LIN {X 0,Y 94.79,Z 775.203,A -85,B 0,C 180,E1 3730.047,E2 3730.047} C_VEL
LIN {X 0,Y 85.286,Z 779.428,A -85,B 0,C 180,E1 3718.728,E2 3718.728} C_VEL
LIN {X 0,Y 79.196,Z 781.917,A -85,B 0,C 180,E1 3705.374,E2 3705.374} C_VEL
LIN {X 0,Y 77.022,Z 782.778,A -85,B 0,C 180,E1 3690.744,E2 3690.744} C_VEL
LIN {X 0,Y 78.595,Z 782.144,A -85,B 0,C 180,E1 3676.763,E2 3676.763} C_VEL
LIN {X 0,Y 84.097,Z 779.929,A -85,B 0,C 180,E1 3663.142,E2 3663.142} C_VEL
LIN {X 0,Y 93.116,Z 776.003,A -85,B 0,C 180,E1 3651.481,E2 3651.481} C_VEL
LIN {X 0,Y 104.314,Z 770.552,A -85,B 0,C 180,E1 3642.436,E2 3642.436} C_VEL
LIN {X 0,Y 117.401,Z 763.276,A -85,B 0,C 180,E1 3635.158,E2 3635.158} C_VEL
LIN {X 0,Y 131.069,Z 754.49,A -85,B 0,C 180,E1 3629.586,E2 3629.586} C_VEL
LIN {X 0,Y 145.656,Z 743.569,A -85,B 0,C 180,E1 3625.03,E2 3625.03} C_VEL
LIN {X 0,Y 159.184,Z 731.747,A -85,B 0,C 180,E1 3621.631,E2 3621.631} C_VEL
LIN {X 0,Y 172.242,Z 718.44,A -85,B 0,C 180,E1 3618.884,E2 3618.884} C_VEL
LIN {X 0,Y 184.101,Z 704.311,A -85,B 0,C 180,E1 3616.73,E2 3616.73} C_VEL
LIN {X 0,Y 195.07,Z 688.928,A -85,B 0,C 180,E1 3614.95,E2 3614.95} C_VEL
LIN {X 0,Y 205.1,Z 672.108,A -85,B 0,C 180,E1 3613.461,E2 3613.461} C_VEL
LIN {X 0,Y 213.82,Z 654.238,A -85,B 0,C 180,E1 3612.234,E2 3612.234} C_VEL
LIN {X 0,Y 220.959,Z 635.839,A -85,B 0,C 180,E1 3611.251,E2 3611.251} C_VEL
LIN {X 0,Y 226.74,Z 615.995,A -85,B 0,C 180,E1 3610.436,E2 3610.436} C_VEL
LIN {X 0,Y 230.757,Z 595.786,A -85,B 0,C 180,E1 3609.81,E2 3609.81} C_VEL
LIN {X 0,Y 236.026,Z 551.57,A -85,B 0,C 180,E1 3608.94,E2 3608.94} C_VEL
LIN {X 0,Y 238.75,Z 528.075,A -85,B 0,C 180,E1 3608.563,E2 3608.563} C_VEL
LIN {X 0,Y 238.273,Z 526.572,A -85,B 0,C 180,E1 3606.506,E2 3606.506} C_VEL
LIN {X 0,Y 237.888,Z 526.562,A -85,B 0,C 180,E1 3602.168,E2 3602.168} C_VEL
LIN {X 0,Y 238.215,Z 528.774,A -85,B 0,C 180,E1 3598.918,E2 3598.918} C_VEL
LIN {X 0,Y 238.522,Z 530.833,A -85,B 0,C 180,E1 3597.356,E2 3597.356} C_VEL
LIN {X 0,Y 229.693,Z 603.415,A -85,B 0,C 180,E1 3596.168,E2 3596.168} C_VEL
LIN {X 0,Y 225.268,Z 624.242,A -85,B 0,C 180,E1 3595.75,E2 3595.75} C_VEL
LIN {X 0,Y 219.212,Z 644.095,A -85,B 0,C 180,E1 3595.261,E2 3595.261} C_VEL
LIN {X 0,Y 211.383,Z 663.553,A -85,B 0,C 180,E1 3594.655,E2 3594.655} C_VEL
LIN {X 0,Y 202.115,Z 681.945,A -85,B 0,C 180,E1 3593.885,E2 3593.885} C_VEL
LIN {X 0,Y 190.896,Z 700.299,A -85,B 0,C 180,E1 3592.779,E2 3592.779} C_VEL
LIN {X 0,Y 178.447,Z 717.368,A -85,B 0,C 180,E1 3591.299,E2 3591.299} C_VEL
LIN {X 0,Y 164.832,Z 733.27,A -85,B 0,C 180,E1 3589.311,E2 3589.311} C_VEL
LIN {X 0,Y 150.054,Z 748.089,A -85,B 0,C 180,E1 3586.61,E2 3586.61} C_VEL
LIN {X 0,Y 134.86,Z 761.302,A -85,B 0,C 180,E1 3583.016,E2 3583.016} C_VEL
LIN {X 0,Y 119.586,Z 772.97,A -85,B 0,C 180,E1 3578.131,E2 3578.131} C_VEL
LIN {X 0,Y 104.755,Z 783.066,A -85,B 0,C 180,E1 3571.412,E2 3571.412} C_VEL
LIN {X 0,Y 91.293,Z 791.543,A -85,B 0,C 180,E1 3562.049,E2 3562.049} C_VEL
LIN {X 0,Y 81.046,Z 798.03,A -85,B 0,C 180,E1 3549.904,E2 3549.904} C_VEL
LIN {X 0,Y 77.511,Z 800.568,A -85,B 0,C 180,E1 3542.778,E2 3542.778} C_VEL
LIN {X 0,Y 74.757,Z 801.989,A -85,B 0,C 180,E1 3537.407,E2 3537.407} C_VEL
LIN {X 0,Y 68.448,Z 803.712,A -85,B 0,C 180,E1 3525.965,E2 3525.965} C_VEL
LIN {X 0,Y 66.797,Z 804.343,A -85,B 0,C 180,E1 3518.037,E2 3518.037} C_VEL
LIN {X 0,Y 66.981,Z 804.481,A -85,B 0,C 180,E1 3515.654,E2 3515.654} C_VEL
LIN {X 0,Y 67.99,Z 804.819,A -85,B 0,C 180,E1 3509.63,E2 3509.63} C_VEL
LIN {X 0,Y 66.248,Z 803.424,A -85,B 0,C 180,E1 3494.237,E2 3494.237} C_VEL
LIN {X 0,Y 69.077,Z 800.295,A -85,B 0,C 180,E1 3477.619,E2 3477.619} C_VEL
LIN {X 0,Y 77.372,Z 795.212,A -85,B 0,C 180,E1 3462.559,E2 3462.559} C_VEL
LIN {X 0,Y 89.824,Z 788.216,A -85,B 0,C 180,E1 3451.009,E2 3451.009} C_VEL
LIN {X 0,Y 104.215,Z 779.674,A -85,B 0,C 180,E1 3442.924,E2 3442.924} C_VEL
LIN {X 0,Y 119.332,Z 769.699,A -85,B 0,C 180,E1 3437.223,E2 3437.223} C_VEL
LIN {X 0,Y 134.489,Z 758.36,A -85,B 0,C 180,E1 3433.12,E2 3433.12} C_VEL
LIN {X 0,Y 149.29,Z 745.693,A -85,B 0,C 180,E1 3430.102,E2 3430.102} C_VEL
LIN {X 0,Y 163.502,Z 731.675,A -85,B 0,C 180,E1 3427.843,E2 3427.843} C_VEL
LIN {X 0,Y 176.979,Z 716.205,A -85,B 0,C 180,E1 3426.12,E2 3426.12} C_VEL
LIN {X 0,Y 189.635,Z 699.109,A -85,B 0,C 180,E1 3424.808,E2 3424.808} C_VEL
LIN {X 0,Y 200.918,Z 680.865,A -85,B 0,C 180,E1 3423.846,E2 3423.846} C_VEL
LIN {X 0,Y 210.287,Z 662.45,A -85,B 0,C 180,E1 3423.175,E2 3423.175} C_VEL
LIN {X 0,Y 218.195,Z 642.954,A -85,B 0,C 180,E1 3422.643,E2 3422.643} C_VEL
LIN {X 0,Y 224.532,Z 622.209,A -85,B 0,C 180,E1 3422.192,E2 3422.192} C_VEL
LIN {X 0,Y 228.935,Z 601.111,A -85,B 0,C 180,E1 3421.809,E2 3421.809} C_VEL
LIN {X 0,Y 236.861,Z 536.432,A -85,B 0,C 180,E1 3420.801,E2 3420.801} C_VEL
LIN {X 0,Y 236.592,Z 534.278,A -85,B 0,C 180,E1 3417.82,E2 3417.82} C_VEL
LIN {X 0,Y 236.945,Z 534.241,A -85,B 0,C 180,E1 3413.701,E2 3413.701} C_VEL
LIN {X 0,Y 237.048,Z 534.547,A -85,B 0,C 180,E1 3413.152,E2 3413.152} C_VEL
LIN {X 0,Y 230.307,Z 591.088,A -85,B 0,C 180,E1 3412.191,E2 3412.191} C_VEL
LIN {X 0,Y 226.826,Z 610.801,A -85,B 0,C 180,E1 3411.658,E2 3411.658} C_VEL
LIN {X 0,Y 221.942,Z 629.319,A -85,B 0,C 180,E1 3411.006,E2 3411.006} C_VEL
LIN {X 0,Y 215.515,Z 647.484,A -85,B 0,C 180,E1 3410.187,E2 3410.187} C_VEL
LIN {X 0,Y 207.188,Z 665.867,A -85,B 0,C 180,E1 3409.123,E2 3409.123} C_VEL
LIN {X 0,Y 197.405,Z 683.311,A -85,B 0,C 180,E1 3407.829,E2 3407.829} C_VEL
LIN {X 0,Y 186.314,Z 699.654,A -85,B 0,C 180,E1 3406.243,E2 3406.243} C_VEL
LIN {X 0,Y 173.527,Z 715.411,A -85,B 0,C 180,E1 3404.201,E2 3404.201} C_VEL
LIN {X 0,Y 160.047,Z 729.424,A -85,B 0,C 180,E1 3401.724,E2 3401.724} C_VEL
LIN {X 0,Y 145.999,Z 741.842,A -85,B 0,C 180,E1 3398.647,E2 3398.647} C_VEL
LIN {X 0,Y 131.542,Z 752.736,A -85,B 0,C 180,E1 3394.756,E2 3394.756} C_VEL
LIN {X 0,Y 116.962,Z 762.108,A -85,B 0,C 180,E1 3389.699,E2 3389.699} C_VEL
LIN {X 0,Y 102.702,Z 769.932,A -85,B 0,C 180,E1 3382.967,E2 3382.967} C_VEL
LIN {X 0,Y 89.463,Z 776.145,A -85,B 0,C 180,E1 3373.861,E2 3373.861} C_VEL
LIN {X 0,Y 78.868,Z 780.452,A -85,B 0,C 180,E1 3362.171,E2 3362.171} C_VEL
LIN {X 0,Y 71.832,Z 783.018,A -85,B 0,C 180,E1 3347.832,E2 3347.832} C_VEL
LIN {X 0,Y 69.156,Z 783.937,A -85,B 0,C 180,E1 3332.486,E2 3332.486} C_VEL
LIN {X 0,Y 70.527,Z 783.466,A -85,B 0,C 180,E1 3316.89,E2 3316.89} C_VEL
LIN {X 0,Y 76.303,Z 781.422,A -85,B 0,C 180,E1 3301.854,E2 3301.854} C_VEL
LIN {X 0,Y 85.91,Z 777.677,A -85,B 0,C 180,E1 3289.328,E2 3289.328} C_VEL
LIN {X 0,Y 98.445,Z 772.088,A -85,B 0,C 180,E1 3279.478,E2 3279.478} C_VEL
LIN {X 0,Y 112.253,Z 764.919,A -85,B 0,C 180,E1 3272.204,E2 3272.204} C_VEL
LIN {X 0,Y 126.523,Z 756.253,A -85,B 0,C 180,E1 3266.752,E2 3266.752} C_VEL
LIN {X 0,Y 140.772,Z 746.14,A -85,B 0,C 180,E1 3262.584,E2 3262.584} C_VEL
LIN {X 0,Y 154.677,Z 734.619,A -85,B 0,C 180,E1 3259.311,E2 3259.311} C_VEL
LIN {X 0,Y 168.049,Z 721.668,A -85,B 0,C 180,E1 3256.687,E2 3256.687} C_VEL
LIN {X 0,Y 180.762,Z 707.191,A -85,B 0,C 180,E1 3254.543,E2 3254.543} C_VEL
LIN {X 0,Y 192.724,Z 690.993,A -85,B 0,C 180,E1 3252.756,E2 3252.756} C_VEL
LIN {X 0,Y 202.946,Z 674.402,A -85,B 0,C 180,E1 3251.366,E2 3251.366} C_VEL
LIN {X 0,Y 211.824,Z 656.824,A -85,B 0,C 180,E1 3250.219,E2 3250.219} C_VEL
LIN {X 0,Y 219.327,Z 638.171,A -85,B 0,C 180,E1 3249.269,E2 3249.269} C_VEL
LIN {X 0,Y 225.338,Z 618.422,A -85,B 0,C 180,E1 3248.491,E2 3248.491} C_VEL
LIN {X 0,Y 229.599,Z 598.14,A -85,B 0,C 180,E1 3247.882,E2 3247.882} C_VEL
LIN {X 0,Y 234.631,Z 557.443,A -85,B 0,C 180,E1 3247.085,E2 3247.085} C_VEL
LIN {X 0,Y 237.333,Z 534.597,A -85,B 0,C 180,E1 3246.714,E2 3246.714} C_VEL
LIN {X 0,Y 236.89,Z 534.461,A -85,B 0,C 180,E1 3242.42,E2 3242.42} C_VEL
LIN {X 0,Y 237.097,Z 536.385,A -85,B 0,C 180,E1 3239.517,E2 3239.517} C_VEL
LIN {X 0,Y 237.127,Z 536.857,A -85,B 0,C 180,E1 3239.187,E2 3239.187} C_VEL
LIN {X 0,Y 228.983,Z 602.568,A -85,B 0,C 180,E1 3238.174,E2 3238.174} C_VEL
LIN {X 0,Y 224.534,Z 623.283,A -85,B 0,C 180,E1 3237.795,E2 3237.795} C_VEL
LIN {X 0,Y 218.444,Z 643.068,A -85,B 0,C 180,E1 3237.363,E2 3237.363} C_VEL
LIN {X 0,Y 210.782,Z 661.997,A -85,B 0,C 180,E1 3236.851,E2 3236.851} C_VEL
LIN {X 0,Y 200.92,Z 681.371,A -85,B 0,C 180,E1 3236.147,E2 3236.147} C_VEL
LIN {X 0,Y 189.637,Z 699.509,A -85,B 0,C 180,E1 3235.184,E2 3235.184} C_VEL
LIN {X 0,Y 176.981,Z 716.533,A -85,B 0,C 180,E1 3233.873,E2 3233.873} C_VEL
LIN {X 0,Y 163.027,Z 732.455,A -85,B 0,C 180,E1 3232.081,E2 3232.081} C_VEL
LIN {X 0,Y 148.356,Z 746.799,A -85,B 0,C 180,E1 3229.72,E2 3229.72} C_VEL
LIN {X 0,Y 132.674,Z 760.024,A -85,B 0,C 180,E1 3226.444,E2 3226.444} C_VEL
LIN {X 0,Y 116.739,Z 771.695,A -85,B 0,C 180,E1 3221.93,E2 3221.93} C_VEL
LIN {X 0,Y 101.029,Z 781.796,A -85,B 0,C 180,E1 3215.571,E2 3215.571} C_VEL
LIN {X 0,Y 86.409,Z 790.275,A -85,B 0,C 180,E1 3206.419,E2 3206.419} C_VEL
LIN {X 0,Y 74.612,Z 796.891,A -85,B 0,C 180,E1 3193.646,E2 3193.646} C_VEL
LIN {X 0,Y 67.665,Z 801.488,A -85,B 0,C 180,E1 3177.556,E2 3177.556} C_VEL
LIN {X 0,Y 66.421,Z 804.095,A -85,B 0,C 180,E1 3160.407,E2 3160.407} C_VEL
LIN {X 0,Y 66.981,Z 804.481,A -85,B 0,C 180,E1 3155.654,E2 3155.654} C_VEL
LIN {X 0,Y 66.693,Z 804.571,A -85,B 0,C 180,E1 3152.598,E2 3152.598} C_VEL
LIN {X 0,Y 64.66,Z 804.284,A -85,B 0,C 180,E1 3148.461,E2 3148.461} C_VEL
LIN {X 0,Y 58.75,Z 802.884,A -85,B 0,C 180,E1 3138.157,E2 3138.157} C_VEL
LIN {X 0,Y 58.309,Z 802.507,A -85,B 0,C 180,E1 3135.107,E2 3135.107} C_VEL
LIN {X 0,Y 61.542,Z 799.446,A -85,B 0,C 180,E1 3115.346,E2 3115.346} C_VEL
LIN {X 0,Y 70.802,Z 794.549,A -85,B 0,C 180,E1 3099.042,E2 3099.042} C_VEL
LIN {X 0,Y 83.558,Z 788.148,A -85,B 0,C 180,E1 3087.692,E2 3087.692} C_VEL
LIN {X 0,Y 99.129,Z 779.667,A -85,B 0,C 180,E1 3079.441,E2 3079.441} C_VEL
LIN {X 0,Y 115.328,Z 769.658,A -85,B 0,C 180,E1 3073.838,E2 3073.838} C_VEL
LIN {X 0,Y 130.975,Z 758.559,A -85,B 0,C 180,E1 3070.019,E2 3070.019} C_VEL
LIN {X 0,Y 147.104,Z 745.276,A -85,B 0,C 180,E1 3067.101,E2 3067.101} C_VEL
LIN {X 0,Y 162.096,Z 730.871,A -85,B 0,C 180,E1 3065.026,E2 3065.026} C_VEL
LIN {X 0,Y 176.293,Z 714.854,A -85,B 0,C 180,E1 3063.469,E2 3063.469} C_VEL
LIN {X 0,Y 189.126,Z 697.707,A -85,B 0,C 180,E1 3062.343,E2 3062.343} C_VEL
LIN {X 0,Y 200.04,Z 680.284,A -85,B 0,C 180,E1 3061.56,E2 3061.56} C_VEL
LIN {X 0,Y 209.496,Z 661.945,A -85,B 0,C 180,E1 3060.993,E2 3060.993} C_VEL
LIN {X 0,Y 217.523,Z 642.437,A -85,B 0,C 180,E1 3060.537,E2 3060.537} C_VEL
LIN {X 0,Y 223.931,Z 621.816,A -85,B 0,C 180,E1 3060.145,E2 3060.145} C_VEL
LIN {X 0,Y 228.431,Z 600.738,A -85,B 0,C 180,E1 3059.801,E2 3059.801} C_VEL
LIN {X 0,Y 235.632,Z 543.029,A -85,B 0,C 180,E1 3058.966,E2 3058.966} C_VEL
LIN {X 0,Y 235.593,Z 542.128,A -85,B 0,C 180,E1 3057.324,E2 3057.324} C_VEL
LIN {X 0,Y 235.733,Z 542.122,A -85,B 0,C 180,E1 3054.985,E2 3054.985} C_VEL
LIN {X 0,Y 229.443,Z 593.572,A -85,B 0,C 180,E1 3054.131,E2 3054.131} C_VEL
LIN {X 0,Y 225.559,Z 614.046,A -85,B 0,C 180,E1 3053.593,E2 3053.593} C_VEL
LIN {X 0,Y 220.134,Z 633.241,A -85,B 0,C 180,E1 3052.937,E2 3052.937} C_VEL
LIN {X 0,Y 212.981,Z 652.126,A -85,B 0,C 180,E1 3052.109,E2 3052.109} C_VEL
LIN {X 0,Y 204.421,Z 669.941,A -85,B 0,C 180,E1 3051.112,E2 3051.112} C_VEL
LIN {X 0,Y 194.523,Z 686.751,A -85,B 0,C 180,E1 3049.916,E2 3049.916} C_VEL
LIN {X 0,Y 183.19,Z 702.748,A -85,B 0,C 180,E1 3048.433,E2 3048.433} C_VEL
LIN {X 0,Y 170.616,Z 717.665,A -85,B 0,C 180,E1 3046.601,E2 3046.601} C_VEL
LIN {X 0,Y 157.746,Z 730.671,A -85,B 0,C 180,E1 3044.453,E2 3044.453} C_VEL
LIN {X 0,Y 143.306,Z 743.076,A -85,B 0,C 180,E1 3041.596,E2 3041.596} C_VEL
LIN {X 0,Y 128.363,Z 753.961,A -85,B 0,C 180,E1 3037.957,E2 3037.957} C_VEL
LIN {X 0,Y 113.169,Z 763.326,A -85,B 0,C 180,E1 3033.166,E2 3033.166} C_VEL
LIN {X 0,Y 97.751,Z 771.333,A -85,B 0,C 180,E1 3026.471,E2 3026.471} C_VEL
LIN {X 0,Y 83.271,Z 777.616,A -85,B 0,C 180,E1 3017.09,E2 3017.09} C_VEL
LIN {X 0,Y 71.46,Z 781.937,A -85,B 0,C 180,E1 3004.355,E2 3004.355} C_VEL
LIN {X 0,Y 63.8,Z 784.403,A -85,B 0,C 180,E1 2988.266,E2 2988.266} C_VEL
LIN {X 0,Y 61.2,Z 785.2,A -85,B 0,C 180,E1 2970,E2 2970} C_VEL
LIN {X 0,Y 63.781,Z 784.429,A -85,B 0,C 180,E1 2951.729,E2 2951.729} C_VEL
LIN {X 0,Y 71.262,Z 782.046,A -85,B 0,C 180,E1 2935.861,E2 2935.861} C_VEL
LIN {X 0,Y 82.576,Z 777.942,A -85,B 0,C 180,E1 2923.408,E2 2923.408} C_VEL
LIN {X 0,Y 95.818,Z 772.302,A -85,B 0,C 180,E1 2914.479,E2 2914.479} C_VEL
LIN {X 0,Y 109.848,Z 765.261,A -85,B 0,C 180,E1 2908.007,E2 2908.007} C_VEL
LIN {X 0,Y 124.866,Z 756.375,A -85,B 0,C 180,E1 2902.952,E2 2902.952} C_VEL
LIN {X 0,Y 139.694,Z 746.022,A -85,B 0,C 180,E1 2899.133,E2 2899.133} C_VEL
LIN {X 0,Y 154.055,Z 734.233,A -85,B 0,C 180,E1 2896.152,E2 2896.152} C_VEL
LIN {X 0,Y 167.795,Z 720.972,A -85,B 0,C 180,E1 2893.77,E2 2893.77} C_VEL
LIN {X 0,Y 180.342,Z 706.72,A -85,B 0,C 180,E1 2891.895,E2 2891.895} C_VEL
LIN {X 0,Y 191.484,Z 691.818,A -85,B 0,C 180,E1 2890.405,E2 2890.405} C_VEL
LIN {X 0,Y 201.999,Z 674.988,A -85,B 0,C 180,E1 2889.114,E2 2889.114} C_VEL
LIN {X 0,Y 211.047,Z 657.306,A -85,B 0,C 180,E1 2888.057,E2 2888.057} C_VEL
LIN {X 0,Y 218.915,Z 637.859,A -85,B 0,C 180,E1 2887.149,E2 2887.149} C_VEL
LIN {X 0,Y 224.94,Z 617.986,A -85,B 0,C 180,E1 2886.432,E2 2886.432} C_VEL
LIN {X 0,Y 229.184,Z 597.547,A -85,B 0,C 180,E1 2885.866,E2 2885.866} C_VEL
LIN {X 0,Y 234.66,Z 553.561,A -85,B 0,C 180,E1 2885.077,E2 2885.077} C_VEL
LIN {X 0,Y 236.022,Z 542.248,A -85,B 0,C 180,E1 2884.901,E2 2884.901} C_VEL
LIN {X 0,Y 235.911,Z 542.576,A -85,B 0,C 180,E1 2881.944,E2 2881.944} C_VEL
LIN {X 0,Y 235.906,Z 543.467,A -85,B 0,C 180,E1 2881.03,E2 2881.03} C_VEL
LIN {X 0,Y 228.524,Z 601.888,A -85,B 0,C 180,E1 2880.186,E2 2880.186} C_VEL
LIN {X 0,Y 224.052,Z 622.45,A -85,B 0,C 180,E1 2879.848,E2 2879.848} C_VEL
LIN {X 0,Y 217.921,Z 642.174,A -85,B 0,C 180,E1 2879.475,E2 2879.475} C_VEL
LIN {X 0,Y 209.994,Z 661.529,A -85,B 0,C 180,E1 2879.027,E2 2879.027} C_VEL
LIN {X 0,Y 200.538,Z 679.92,A -85,B 0,C 180,E1 2878.464,E2 2878.464} C_VEL
LIN {X 0,Y 189.127,Z 698.131,A -85,B 0,C 180,E1 2877.649,E2 2877.649} C_VEL
LIN {X 0,Y 176.294,Z 715.199,A -85,B 0,C 180,E1 2876.523,E2 2876.523} C_VEL
LIN {X 0,Y 162.585,Z 730.642,A -85,B 0,C 180,E1 2875.025,E2 2875.025} C_VEL
LIN {X 0,Y 147.106,Z 745.507,A -85,B 0,C 180,E1 2872.891,E2 2872.891} C_VEL
LIN {X 0,Y 130.978,Z 758.744,A -85,B 0,C 180,E1 2869.975,E2 2869.975} C_VEL
LIN {X 0,Y 114.43,Z 770.421,A -85,B 0,C 180,E1 2865.897,E2 2865.897} C_VEL
LIN {X 0,Y 97.874,Z 780.525,A -85,B 0,C 180,E1 2860.022,E2 2860.022} C_VEL
LIN {X 0,Y 82.085,Z 789.006,A -85,B 0,C 180,E1 2851.282,E2 2851.282} C_VEL
LIN {X 0,Y 69.092,Z 795.5,A -85,B 0,C 180,E1 2838.806,E2 2838.806} C_VEL
LIN {X 0,Y 60.631,Z 800.105,A -85,B 0,C 180,E1 2821.849,E2 2821.849} C_VEL
LIN {X 0,Y 58.387,Z 802.851,A -85,B 0,C 180,E1 2801.858,E2 2801.858} C_VEL
LIN {X 0,Y 59.99,Z 803.61,A -85,B 0,C 180,E1 2789.92,E2 2789.92} C_VEL
LIN {X 0,Y 58.309,Z 802.507,A -85,B 0,C 180,E1 2775.107,E2 2775.107} C_VEL
LIN {X 0,Y 57.755,Z 801.514,A -85,B 0,C 180,E1 2767.524,E2 2767.524} C_VEL
LIN {X 0,Y 57.592,Z 797.296,A -85,B 0,C 180,E1 2746.102,E2 2746.102} C_VEL
LIN {X 0,Y 59.976,Z 795.854,A -85,B 0,C 180,E1 2740.775,E2 2740.775} C_VEL
LIN {X 0,Y 72.988,Z 790.122,A -85,B 0,C 180,E1 2727.075,E2 2727.075} C_VEL
LIN {X 0,Y 88.363,Z 782.767,A -85,B 0,C 180,E1 2718.11,E2 2718.11} C_VEL
LIN {X 0,Y 104.879,Z 773.742,A -85,B 0,C 180,E1 2712.106,E2 2712.106} C_VEL
LIN {X 0,Y 121.175,Z 763.407,A -85,B 0,C 180,E1 2708.053,E2 2708.053} C_VEL
LIN {X 0,Y 137.53,Z 751.311,A -85,B 0,C 180,E1 2705.139,E2 2705.139} C_VEL
LIN {X 0,Y 153.668,Z 737.323,A -85,B 0,C 180,E1 2702.983,E2 2702.983} C_VEL
LIN {X 0,Y 168.442,Z 722.251,A -85,B 0,C 180,E1 2701.454,E2 2701.454} C_VEL
LIN {X 0,Y 181.972,Z 705.964,A -85,B 0,C 180,E1 2700.349,E2 2700.349} C_VEL
LIN {X 0,Y 193.973,Z 688.764,A -85,B 0,C 180,E1 2699.563,E2 2699.563} C_VEL
LIN {X 0,Y 204.496,Z 670.555,A -85,B 0,C 180,E1 2699.006,E2 2699.006} C_VEL
LIN {X 0,Y 213.528,Z 651.227,A -85,B 0,C 180,E1 2698.59,E2 2698.59} C_VEL
LIN {X 0,Y 220.816,Z 631.121,A -85,B 0,C 180,E1 2698.242,E2 2698.242} C_VEL
LIN {X 0,Y 226.297,Z 610.268,A -85,B 0,C 180,E1 2697.927,E2 2697.927} C_VEL
LIN {X 0,Y 229.862,Z 588.948,A -85,B 0,C 180,E1 2697.629,E2 2697.629} C_VEL
LIN {X 0,Y 234.62,Z 550.029,A -85,B 0,C 180,E1 2697.068,E2 2697.068} C_VEL
LIN {X 0,Y 234.603,Z 550.172,A -85,B 0,C 180,E1 2696.831,E2 2696.831} C_VEL
LIN {X 0,Y 228.774,Z 596.534,A -85,B 0,C 180,E1 2696.072,E2 2696.072} C_VEL
LIN {X 0,Y 224.789,Z 616.292,A -85,B 0,C 180,E1 2695.574,E2 2695.574} C_VEL
LIN {X 0,Y 219.306,Z 634.998,A -85,B 0,C 180,E1 2694.974,E2 2694.974} C_VEL
LIN {X 0,Y 212.044,Z 653.683,A -85,B 0,C 180,E1 2694.214,E2 2694.214} C_VEL
LIN {X 0,Y 202.871,Z 672.256,A -85,B 0,C 180,E1 2693.253,E2 2693.253} C_VEL
LIN {X 0,Y 192.291,Z 689.613,A -85,B 0,C 180,E1 2692.104,E2 2692.104} C_VEL
LIN {X 0,Y 180.343,Z 705.825,A -85,B 0,C 180,E1 2690.695,E2 2690.695} C_VEL
LIN {X 0,Y 167.071,Z 720.899,A -85,B 0,C 180,E1 2688.948,E2 2688.948} C_VEL
LIN {X 0,Y 152.678,Z 734.658,A -85,B 0,C 180,E1 2686.749,E2 2686.749} C_VEL
LIN {X 0,Y 137.345,Z 747.003,A -85,B 0,C 180,E1 2683.929,E2 2683.929} C_VEL
LIN {X 0,Y 121.154,Z 757.938,A -85,B 0,C 180,E1 2680.185,E2 2680.185} C_VEL
LIN {X 0,Y 105.121,Z 766.97,A -85,B 0,C 180,E1 2675.258,E2 2675.258} C_VEL
LIN {X 0,Y 89.249,Z 774.383,A -85,B 0,C 180,E1 2668.365,E2 2668.365} C_VEL
LIN {X 0,Y 74.638,Z 780.002,A -85,B 0,C 180,E1 2658.604,E2 2658.604} C_VEL
LIN {X 0,Y 62.804,Z 783.772,A -85,B 0,C 180,E1 2644.968,E2 2644.968} C_VEL
LIN {X 0,Y 55.242,Z 785.846,A -85,B 0,C 180,E1 2626.833,E2 2626.833} C_VEL
LIN {X 0,Y 53.351,Z 786.348,A -85,B 0,C 180,E1 2606.777,E2 2606.777} C_VEL
LIN {X 0,Y 56.942,Z 785.467,A -85,B 0,C 180,E1 2587.276,E2 2587.276} C_VEL
LIN {X 0,Y 65.952,Z 782.941,A -85,B 0,C 180,E1 2570.453,E2 2570.453} C_VEL
LIN {X 0,Y 78.749,Z 778.667,A -85,B 0,C 180,E1 2558.078,E2 2558.078} C_VEL
LIN {X 0,Y 93.957,Z 772.498,A -85,B 0,C 180,E1 2549.24,E2 2549.24} C_VEL
LIN {X 0,Y 109.988,Z 764.604,A -85,B 0,C 180,E1 2543.011,E2 2543.011} C_VEL
LIN {X 0,Y 126.173,Z 754.999,A -85,B 0,C 180,E1 2538.481,E2 2538.481} C_VEL
LIN {X 0,Y 141.882,Z 743.858,A -85,B 0,C 180,E1 2535.11,E2 2535.11} C_VEL
LIN {X 0,Y 156.749,Z 731.349,A -85,B 0,C 180,E1 2532.526,E2 2532.526} C_VEL
LIN {X 0,Y 171.051,Z 717.058,A -85,B 0,C 180,E1 2530.441,E2 2530.441} C_VEL
LIN {X 0,Y 184.125,Z 701.487,A -85,B 0,C 180,E1 2528.778,E2 2528.778} C_VEL
LIN {X 0,Y 195.624,Z 685.09,A -85,B 0,C 180,E1 2527.464,E2 2527.464} C_VEL
LIN {X 0,Y 205.693,Z 667.69,A -85,B 0,C 180,E1 2526.389,E2 2526.389} C_VEL
LIN {X 0,Y 214.444,Z 648.925,A -85,B 0,C 180,E1 2525.481,E2 2525.481} C_VEL
LIN {X 0,Y 221.561,Z 629.164,A -85,B 0,C 180,E1 2524.733,E2 2524.733} C_VEL
LIN {X 0,Y 226.833,Z 608.925,A -85,B 0,C 180,E1 2524.135,E2 2524.135} C_VEL
LIN {X 0,Y 230.244,Z 588.417,A -85,B 0,C 180,E1 2523.668,E2 2523.668} C_VEL
LIN {X 0,Y 234.909,Z 550.241,A -85,B 0,C 180,E1 2523.05,E2 2523.05} C_VEL
LIN {X 0,Y 234.874,Z 550.537,A -85,B 0,C 180,E1 2522.885,E2 2522.885} C_VEL
LIN {X 0,Y 228.383,Z 601.024,A -85,B 0,C 180,E1 2522.206,E2 2522.206} C_VEL
LIN {X 0,Y 223.867,Z 621.585,A -85,B 0,C 180,E1 2521.909,E2 2521.909} C_VEL
LIN {X 0,Y 217.741,Z 641.16,A -85,B 0,C 180,E1 2521.596,E2 2521.596} C_VEL
LIN {X 0,Y 210.013,Z 659.968,A -85,B 0,C 180,E1 2521.24,E2 2521.24} C_VEL
LIN {X 0,Y 200.347,Z 678.704,A -85,B 0,C 180,E1 2520.778,E2 2520.778} C_VEL
LIN {X 0,Y 188.968,Z 696.743,A -85,B 0,C 180,E1 2520.12,E2 2520.12} C_VEL
LIN {X 0,Y 175.988,Z 713.859,A -85,B 0,C 180,E1 2519.186,E2 2519.186} C_VEL
LIN {X 0,Y 161.571,Z 729.855,A -85,B 0,C 180,E1 2517.873,E2 2517.873} C_VEL
LIN {X 0,Y 146.112,Z 744.389,A -85,B 0,C 180,E1 2516.077,E2 2516.077} C_VEL
LIN {X 0,Y 129.791,Z 757.463,A -85,B 0,C 180,E1 2513.583,E2 2513.583} C_VEL
LIN {X 0,Y 112.691,Z 769.146,A -85,B 0,C 180,E1 2510.004,E2 2510.004} C_VEL
LIN {X 0,Y 95.347,Z 779.255,A -85,B 0,C 180,E1 2504.738,E2 2504.738} C_VEL
LIN {X 0,Y 78.415,Z 787.738,A -85,B 0,C 180,E1 2496.64,E2 2496.64} C_VEL
LIN {X 0,Y 63.911,Z 794.235,A -85,B 0,C 180,E1 2484.438,E2 2484.438} C_VEL
LIN {X 0,Y 53.764,Z 798.845,A -85,B 0,C 180,E1 2466.519,E2 2466.519} C_VEL
LIN {X 0,Y 50.391,Z 801.627,A -85,B 0,C 180,E1 2443.538,E2 2443.538} C_VEL
LIN {X 0,Y 51.916,Z 802.384,A -85,B 0,C 180,E1 2430,E2 2430} C_VEL
LIN {X 0,Y 50.587,Z 800.922,A -85,B 0,C 180,E1 2409.16,E2 2409.16} C_VEL
LIN {X 0,Y 56.209,Z 797.564,A -85,B 0,C 180,E1 2387.473,E2 2387.473} C_VEL
LIN {X 0,Y 59.976,Z 795.854,A -85,B 0,C 180,E1 2380.775,E2 2380.775} C_VEL
LIN {X 0,Y 63.488,Z 793.944,A -85,B 0,C 180,E1 2374.597,E2 2374.597} C_VEL
LIN {X 0,Y 73.141,Z 787.653,A -85,B 0,C 180,E1 2359.522,E2 2359.522} C_VEL
LIN {X 0,Y 77.807,Z 785.332,A -85,B 0,C 180,E1 2356.368,E2 2356.368} C_VEL
LIN {X 0,Y 94.429,Z 777.363,A -85,B 0,C 180,E1 2350.037,E2 2350.037} C_VEL
LIN {X 0,Y 111.547,Z 767.711,A -85,B 0,C 180,E1 2345.775,E2 2345.775} C_VEL
LIN {X 0,Y 129.127,Z 755.981,A -85,B 0,C 180,E1 2342.751,E2 2342.751} C_VEL
LIN {X 0,Y 145.985,Z 742.671,A -85,B 0,C 180,E1 2340.653,E2 2340.653} C_VEL
LIN {X 0,Y 161.488,Z 728.226,A -85,B 0,C 180,E1 2339.199,E2 2339.199} C_VEL
LIN {X 0,Y 175.559,Z 712.766,A -85,B 0,C 180,E1 2338.173,E2 2338.173} C_VEL
LIN {X 0,Y 188.154,Z 696.372,A -85,B 0,C 180,E1 2337.452,E2 2337.452} C_VEL
LIN {X 0,Y 199.249,Z 679.077,A -85,B 0,C 180,E1 2336.947,E2 2336.947} C_VEL
LIN {X 0,Y 208.833,Z 660.918,A -85,B 0,C 180,E1 2336.594,E2 2336.594} C_VEL
LIN {X 0,Y 212.676,Z 652.363,A -85,B 0,C 180,E1 2336.453,E2 2336.453} C_VEL
LIN {X 0,Y 204.053,Z 670.181,A -85,B 0,C 180,E1 2335.652,E2 2335.652} C_VEL
LIN {X 0,Y 193.664,Z 687.596,A -85,B 0,C 180,E1 2334.667,E2 2334.667} C_VEL
LIN {X 0,Y 182.141,Z 703.588,A -85,B 0,C 180,E1 2333.496,E2 2333.496} C_VEL
LIN {X 0,Y 169.105,Z 718.73,A -85,B 0,C 180,E1 2332.031,E2 2332.031} C_VEL
LIN {X 0,Y 155.214,Z 732.323,A -85,B 0,C 180,E1 2330.254,E2 2330.254} C_VEL
LIN {X 0,Y 140.061,Z 744.825,A -85,B 0,C 180,E1 2327.954,E2 2327.954} C_VEL
LIN {X 0,Y 124.215,Z 755.806,A -85,B 0,C 180,E1 2324.995,E2 2324.995} C_VEL
LIN {X 0,Y 107.843,Z 765.272,A -85,B 0,C 180,E1 2321.025,E2 2321.025} C_VEL
LIN {X 0,Y 91.236,Z 773.187,A -85,B 0,C 180,E1 2315.447,E2 2315.447} C_VEL
LIN {X 0,Y 75.702,Z 779.207,A -85,B 0,C 180,E1 2307.702,E2 2307.702} C_VEL
LIN {X 0,Y 61.349,Z 783.693,A -85,B 0,C 180,E1 2295.814,E2 2295.814} C_VEL
LIN {X 0,Y 50.55,Z 786.423,A -85,B 0,C 180,E1 2278.34,E2 2278.34} C_VEL
LIN {X 0,Y 45.608,Z 787.501,A -85,B 0,C 180,E1 2256.293,E2 2256.293} C_VEL
LIN {X 0,Y 47.165,Z 787.194,A -85,B 0,C 180,E1 2232.736,E2 2232.736} C_VEL
LIN {X 0,Y 55.349,Z 785.326,A -85,B 0,C 180,E1 2212.108,E2 2212.108} C_VEL
LIN {X 0,Y 67.439,Z 782.004,A -85,B 0,C 180,E1 2198.209,E2 2198.209} C_VEL
LIN {X 0,Y 82.847,Z 776.709,A -85,B 0,C 180,E1 2188.239,E2 2188.239} C_VEL
LIN {X 0,Y 98.957,Z 769.858,A -85,B 0,C 180,E1 2181.638,E2 2181.638} C_VEL
LIN {X 0,Y 115.928,Z 761.002,A -85,B 0,C 180,E1 2176.799,E2 2176.799} C_VEL
LIN {X 0,Y 132.531,Z 750.496,A -85,B 0,C 180,E1 2173.296,E2 2173.296} C_VEL
LIN {X 0,Y 147.58,Z 739.153,A -85,B 0,C 180,E1 2170.78,E2 2170.78} C_VEL
LIN {X 0,Y 162.832,Z 725.464,A -85,B 0,C 180,E1 2168.668,E2 2168.668} C_VEL
LIN {X 0,Y 176.794,Z 710.501,A -85,B 0,C 180,E1 2167.017,E2 2167.017} C_VEL
LIN {X 0,Y 189.401,Z 694.329,A -85,B 0,C 180,E1 2165.691,E2 2165.691} C_VEL
LIN {X 0,Y 200.614,Z 676.933,A -85,B 0,C 180,E1 2164.607,E2 2164.607} C_VEL
LIN {X 0,Y 209.954,Z 659.194,A -85,B 0,C 180,E1 2163.74,E2 2163.74} C_VEL
LIN {X 0,Y 212.304,Z 653.923,A -85,B 0,C 180,E1 2163.519,E2 2163.519} C_VEL
LIN {X 0,Y 203.282,Z 672.394,A -85,B 0,C 180,E1 2163.202,E2 2163.202} C_VEL
LIN {X 0,Y 192.691,Z 690.076,A -85,B 0,C 180,E1 2162.762,E2 2162.762} C_VEL
LIN {X 0,Y 180.67,Z 706.774,A -85,B 0,C 180,E1 2162.133,E2 2162.133} C_VEL
LIN {X 0,Y 167.642,Z 722.073,A -85,B 0,C 180,E1 2161.274,E2 2161.274} C_VEL
LIN {X 0,Y 152.974,Z 736.714,A -85,B 0,C 180,E1 2160.04,E2 2160.04} C_VEL
LIN {X 0,Y 137.036,Z 750.232,A -85,B 0,C 180,E1 2158.303,E2 2158.303} C_VEL
LIN {X 0,Y 120.293,Z 762.301,A -85,B 0,C 180,E1 2155.86,E2 2155.86} C_VEL
LIN {X 0,Y 102.399,Z 773.217,A -85,B 0,C 180,E1 2152.144,E2 2152.144} C_VEL
LIN {X 0,Y 84.326,Z 782.486,A -85,B 0,C 180,E1 2146.471,E2 2146.471} C_VEL
LIN {X 0,Y 67.139,Z 789.96,A -85,B 0,C 180,E1 2137.413,E2 2137.413} C_VEL
LIN {X 0,Y 52.493,Z 795.592,A -85,B 0,C 180,E1 2122.449,E2 2122.449} C_VEL
LIN {X 0,Y 43.546,Z 799.345,A -85,B 0,C 180,E1 2098.827,E2 2098.827} C_VEL
LIN {X 0,Y 43.371,Z 801.043,A -85,B 0,C 180,E1 2072.642,E2 2072.642} C_VEL
LIN {X 0,Y 43.798,Z 801.151,A -85,B 0,C 180,E1 2070,E2 2070} C_VEL
LIN {X 0,Y 42.989,Z 799.656,A -85,B 0,C 180,E1 2045.099,E2 2045.099} C_VEL
LIN {X 0,Y 50.39,Z 796.299,A -85,B 0,C 180,E1 2021.063,E2 2021.063} C_VEL
LIN {X 0,Y 63.995,Z 791.093,A -85,B 0,C 180,E1 2004.949,E2 2004.949} C_VEL
LIN {X 0,Y 77.807,Z 785.332,A -85,B 0,C 180,E1 1996.368,E2 1996.368} C_VEL
LIN {X 0,Y 83.405,Z 782.539,A -85,B 0,C 180,E1 1993.103,E2 1993.103} C_VEL
LIN {X 0,Y 96.694,Z 774.657,A -85,B 0,C 180,E1 1984.844,E2 1984.844} C_VEL
LIN {X 0,Y 102.777,Z 771.132,A -85,B 0,C 180,E1 1982.957,E2 1982.957} C_VEL
LIN {X 0,Y 119.98,Z 760.841,A -85,B 0,C 180,E1 1980.179,E2 1980.179} C_VEL
LIN {X 0,Y 137.042,Z 748.732,A -85,B 0,C 180,E1 1978.227,E2 1978.227} C_VEL
LIN {X 0,Y 153.203,Z 735.16,A -85,B 0,C 180,E1 1976.867,E2 1976.867} C_VEL
LIN {X 0,Y 168.403,Z 720.049,A -85,B 0,C 180,E1 1975.895,E2 1975.895} C_VEL
LIN {X 0,Y 176.106,Z 711.289,A -85,B 0,C 180,E1 1975.477,E2 1975.477} C_VEL
LIN {X 0,Y 161.85,Z 726.387,A -85,B 0,C 180,E1 1974.033,E2 1974.033} C_VEL
LIN {X 0,Y 146.33,Z 740.113,A -85,B 0,C 180,E1 1972.197,E2 1972.197} C_VEL
LIN {X 0,Y 130.009,Z 752.149,A -85,B 0,C 180,E1 1969.86,E2 1969.86} C_VEL
LIN {X 0,Y 112.984,Z 762.559,A -85,B 0,C 180,E1 1966.761,E2 1966.761} C_VEL
LIN {X 0,Y 95.439,Z 771.333,A -85,B 0,C 180,E1 1962.425,E2 1962.425} C_VEL
LIN {X 0,Y 77.711,Z 778.429,A -85,B 0,C 180,E1 1955.992,E2 1955.992} C_VEL
LIN {X 0,Y 61.329,Z 783.568,A -85,B 0,C 180,E1 1946.248,E2 1946.248} C_VEL
LIN {X 0,Y 47.545,Z 786.903,A -85,B 0,C 180,E1 1930.686,E2 1930.686} C_VEL
LIN {X 0,Y 38.855,Z 788.556,A -85,B 0,C 180,E1 1906.443,E2 1906.443} C_VEL
LIN {X 0,Y 38.196,Z 788.652,A -85,B 0,C 180,E1 1877.913,E2 1877.913} C_VEL
LIN {X 0,Y 45.257,Z 787.359,A -85,B 0,C 180,E1 1853.382,E2 1853.382} C_VEL
LIN {X 0,Y 58.267,Z 784.401,A -85,B 0,C 180,E1 1836.246,E2 1836.246} C_VEL
LIN {X 0,Y 74.593,Z 779.556,A -85,B 0,C 180,E1 1825.402,E2 1825.402} C_VEL
LIN {X 0,Y 91.785,Z 773.007,A -85,B 0,C 180,E1 1818.611,E2 1818.611} C_VEL
LIN {X 0,Y 109.214,Z 764.709,A -85,B 0,C 180,E1 1813.974,E2 1813.974} C_VEL
LIN {X 0,Y 126.169,Z 754.817,A -85,B 0,C 180,E1 1810.692,E2 1810.692} C_VEL
LIN {X 0,Y 142.446,Z 743.362,A -85,B 0,C 180,E1 1808.24,E2 1808.24} C_VEL
LIN {X 0,Y 157.935,Z 730.32,A -85,B 0,C 180,E1 1806.328,E2 1806.328} C_VEL
LIN {X 0,Y 172.574,Z 715.584,A -85,B 0,C 180,E1 1804.792,E2 1804.792} C_VEL
LIN {X 0,Y 175.867,Z 711.955,A -85,B 0,C 180,E1 1804.476,E2 1804.476} C_VEL
LIN {X 0,Y 161.304,Z 727.727,A -85,B 0,C 180,E1 1803.673,E2 1803.673} C_VEL
LIN {X 0,Y 145.112,Z 742.471,A -85,B 0,C 180,E1 1802.493,E2 1802.493} C_VEL
LIN {X 0,Y 127.991,Z 755.597,A -85,B 0,C 180,E1 1800.809,E2 1800.809} C_VEL
LIN {X 0,Y 110.028,Z 767.168,A -85,B 0,C 180,E1 1798.333,E2 1798.333} C_VEL
LIN {X 0,Y 91.401,Z 777.171,A -85,B 0,C 180,E1 1794.527,E2 1794.527} C_VEL
LIN {X 0,Y 73.412,Z 785.202,A -85,B 0,C 180,E1 1788.694,E2 1788.694} C_VEL
LIN {X 0,Y 55.883,Z 791.703,A -85,B 0,C 180,E1 1778.489,E2 1778.489} C_VEL
LIN {X 0,Y 41.04,Z 796.501,A -85,B 0,C 180,E1 1759.045,E2 1759.045} C_VEL
LIN {X 0,Y 34.523,Z 799.286,A -85,B 0,C 180,E1 1727.121,E2 1727.121} C_VEL
LIN {X 0,Y 35.661,Z 799.914,A -85,B 0,C 180,E1 1710,E2 1710} C_VEL
LIN {X 0,Y 35.902,Z 798.299,A -85,B 0,C 180,E1 1678.053,E2 1678.053} C_VEL
LIN {X 0,Y 46.034,Z 794.827,A -85,B 0,C 180,E1 1652.107,E2 1652.107} C_VEL
LIN {X 0,Y 61.78,Z 789.533,A -85,B 0,C 180,E1 1637.284,E2 1637.284} C_VEL
LIN {X 0,Y 78.994,Z 782.724,A -85,B 0,C 180,E1 1629.158,E2 1629.158} C_VEL
LIN {X 0,Y 97.233,Z 774.068,A -85,B 0,C 180,E1 1624.101,E2 1624.101} C_VEL
LIN {X 0,Y 102.777,Z 771.132,A -85,B 0,C 180,E1 1622.957,E2 1622.957} C_VEL
LIN {X 0,Y 108.91,Z 767.484,A -85,B 0,C 180,E1 1621.302,E2 1621.302} C_VEL
LIN {X 0,Y 123.429,Z 757.685,A -85,B 0,C 180,E1 1616.388,E2 1616.388} C_VEL
LIN {X 0,Y 129.469,Z 753.349,A -85,B 0,C 180,E1 1615.395,E2 1615.395} C_VEL
LIN {X 0,Y 139.565,Z 745.837,A -85,B 0,C 180,E1 1614.64,E2 1614.64} C_VEL
LIN {X 0,Y 122.874,Z 757.133,A -85,B 0,C 180,E1 1612.518,E2 1612.518} C_VEL
LIN {X 0,Y 105.684,Z 766.726,A -85,B 0,C 180,E1 1609.704,E2 1609.704} C_VEL
LIN {X 0,Y 88.66,Z 774.461,A -85,B 0,C 180,E1 1605.892,E2 1605.892} C_VEL
LIN {X 0,Y 70.329,Z 781.056,A -85,B 0,C 180,E1 1599.766,E2 1599.766} C_VEL
LIN {X 0,Y 53.172,Z 785.723,A -85,B 0,C 180,E1 1589.879,E2 1589.879} C_VEL
LIN {X 0,Y 38.581,Z 788.624,A -85,B 0,C 180,E1 1572.361,E2 1572.361} C_VEL
LIN {X 0,Y 30.097,Z 789.884,A -85,B 0,C 180,E1 1541.498,E2 1541.498} C_VEL
LIN {X 0,Y 32.014,Z 789.659,A -85,B 0,C 180,E1 1506.046,E2 1506.046} C_VEL
LIN {X 0,Y 43.22,Z 787.88,A -85,B 0,C 180,E1 1480.235,E2 1480.235} C_VEL
LIN {X 0,Y 58.957,Z 784.417,A -85,B 0,C 180,E1 1466,E2 1466} C_VEL
LIN {X 0,Y 76.625,Z 779.126,A -85,B 0,C 180,E1 1457.726,E2 1457.726} C_VEL
LIN {X 0,Y 94.268,Z 772.282,A -85,B 0,C 180,E1 1452.637,E2 1452.637} C_VEL
LIN {X 0,Y 112.376,Z 763.438,A -85,B 0,C 180,E1 1449.037,E2 1449.037} C_VEL
LIN {X 0,Y 129.806,Z 752.952,A -85,B 0,C 180,E1 1446.476,E2 1446.476} C_VEL
LIN {X 0,Y 139.027,Z 746.499,A -85,B 0,C 180,E1 1445.314,E2 1445.314} C_VEL
LIN {X 0,Y 122.272,Z 758.394,A -85,B 0,C 180,E1 1443.965,E2 1443.965} C_VEL
LIN {X 0,Y 105.047,Z 768.698,A -85,B 0,C 180,E1 1442.011,E2 1442.011} C_VEL
LIN {X 0,Y 86.005,Z 778.161,A -85,B 0,C 180,E1 1438.764,E2 1438.764} C_VEL
LIN {X 0,Y 67.414,Z 785.69,A -85,B 0,C 180,E1 1433.559,E2 1433.559} C_VEL
LIN {X 0,Y 48.944,Z 791.712,A -85,B 0,C 180,E1 1423.763,E2 1423.763} C_VEL
LIN {X 0,Y 32.862,Z 796.042,A -85,B 0,C 180,E1 1402.282,E2 1402.282} C_VEL
LIN {X 0,Y 26.624,Z 798.324,A -85,B 0,C 180,E1 1362.486,E2 1362.486} C_VEL
LIN {X 0,Y 27.502,Z 798.675,A -85,B 0,C 180,E1 1350,E2 1350} C_VEL
LIN {X 0,Y 29.488,Z 796.969,A -85,B 0,C 180,E1 1308.236,E2 1308.236} C_VEL
LIN {X 0,Y 43.011,Z 793.354,A -85,B 0,C 180,E1 1281.589,E2 1281.589} C_VEL
LIN {X 0,Y 60.769,Z 787.961,A -85,B 0,C 180,E1 1269.182,E2 1269.182} C_VEL
LIN {X 0,Y 79.084,Z 781.053,A -85,B 0,C 180,E1 1262.849,E2 1262.849} C_VEL
LIN {X 0,Y 97.998,Z 772.289,A -85,B 0,C 180,E1 1259.022,E2 1259.022} C_VEL
LIN {X 0,Y 116.181,Z 762.063,A -85,B 0,C 180,E1 1256.634,E2 1256.634} C_VEL
LIN {X 0,Y 129.469,Z 753.349,A -85,B 0,C 180,E1 1255.395,E2 1255.395} C_VEL
LIN {X 0,Y 127.987,Z 754.261,A -85,B 0,C 180,E1 1254.947,E2 1254.947} C_VEL
LIN {X 0,Y 119.86,Z 759.395,A -85,B 0,C 180,E1 1254.356,E2 1254.356} C_VEL
LIN {X 0,Y 103.567,Z 768.51,A -85,B 0,C 180,E1 1254.171,E2 1254.171} C_VEL
LIN {X 0,Y 92.21,Z 774.105,A -85,B 0,C 180,E1 1254.891,E2 1254.891} C_VEL
LIN {X 0,Y 72.025,Z 782.574,A -85,B 0,C 180,E1 1258.157,E2 1258.157} C_VEL
LIN {X 0,Y 51.512,Z 789.275,A -85,B 0,C 180,E1 1264.451,E2 1264.451} C_VEL
LIN {X 0,Y 32.649,Z 793.94,A -85,B 0,C 180,E1 1278.318,E2 1278.318} C_VEL
LIN {X 0,Y 19.334,Z 796.785,A -85,B 0,C 180,E1 1318.859,E2 1318.859} C_VEL
LIN {X 0,Y 19.33,Z 797.434,A -85,B 0,C 180,E1 1349.999,E2 1349.999} C_VEL
LIN {X 0,Y 24.183,Z 795.689,A -85,B 0,C 180,E1 1405.779,E2 1405.779} C_VEL
LIN {X 0,Y 40.689,Z 792.136,A -85,B 0,C 180,E1 1429.387,E2 1429.387} C_VEL
LIN {X 0,Y 60.005,Z 786.763,A -85,B 0,C 180,E1 1438.711,E2 1438.711} C_VEL
LIN {X 0,Y 79.109,Z 779.885,A -85,B 0,C 180,E1 1443.191,E2 1443.191} C_VEL
LIN {X 0,Y 98.515,Z 771.143,A -85,B 0,C 180,E1 1445.826,E2 1445.826} C_VEL
LIN {X 0,Y 102.59,Z 769.098,A -85,B 0,C 180,E1 1446.241,E2 1446.241} C_VEL
LIN {X 0,Y 84.16,Z 776.957,A -85,B 0,C 180,E1 1449.583,E2 1449.583} C_VEL
LIN {X 0,Y 65.164,Z 783.216,A -85,B 0,C 180,E1 1454.846,E2 1454.846} C_VEL
LIN {X 0,Y 47.012,Z 787.573,A -85,B 0,C 180,E1 1463.865,E2 1463.865} C_VEL
LIN {X 0,Y 30.989,Z 790.177,A -85,B 0,C 180,E1 1482.092,E2 1482.092} C_VEL
LIN {X 0,Y 21.979,Z 791.134,A -85,B 0,C 180,E1 1519.516,E2 1519.516} C_VEL
LIN {X 0,Y 26.02,Z 790.716,A -85,B 0,C 180,E1 1565.197,E2 1565.197} C_VEL
LIN {X 0,Y 40.231,Z 788.736,A -85,B 0,C 180,E1 1590.438,E2 1590.438} C_VEL
LIN {X 0,Y 57.781,Z 785.064,A -85,B 0,C 180,E1 1602.122,E2 1602.122} C_VEL
LIN {X 0,Y 75.563,Z 779.885,A -85,B 0,C 180,E1 1608.28,E2 1608.28} C_VEL
LIN {X 0,Y 93.841,Z 772.906,A -85,B 0,C 180,E1 1612.253,E2 1612.253} C_VEL
LIN {X 0,Y 102.592,Z 768.942,A -85,B 0,C 180,E1 1613.754,E2 1613.754} C_VEL
LIN {X 0,Y 92.21,Z 774.105,A -85,B 0,C 180,E1 1614.891,E2 1614.891} C_VEL
LIN {X 0,Y 84.152,Z 777.602,A -85,B 0,C 180,E1 1615.308,E2 1615.308} C_VEL
LIN {X 0,Y 73.515,Z 781.417,A -85,B 0,C 180,E1 1614.359,E2 1614.359} C_VEL
LIN {X 0,Y 55.026,Z 786.476,A -85,B 0,C 180,E1 1609.629,E2 1609.629} C_VEL
LIN {X 0,Y 54.43,Z 786.622,A -85,B 0,C 180,E1 1609.434,E2 1609.434} C_VEL
LIN {X 0,Y 36.055,Z 790.087,A -85,B 0,C 180,E1 1600.537,E2 1600.537} C_VEL
LIN {X 0,Y 19.375,Z 791.979,A -85,B 0,C 180,E1 1576.259,E2 1576.259} C_VEL
LIN {X 0,Y 14.568,Z 792.315,A -85,B 0,C 180,E1 1509.932,E2 1509.932} C_VEL
LIN {X 0,Y 28.04,Z 791.175,A -85,B 0,C 180,E1 1466.946,E2 1466.946} C_VEL
LIN {X 0,Y 46.287,Z 788.398,A -85,B 0,C 180,E1 1453.582,E2 1453.582} C_VEL
LIN {X 0,Y 65.449,Z 783.885,A -85,B 0,C 180,E1 1447.462,E2 1447.462} C_VEL
LIN {X 0,Y 45.055,Z 789.688,A -85,B 0,C 180,E1 1443.031,E2 1443.031} C_VEL
LIN {X 0,Y 25.282,Z 793.681,A -85,B 0,C 180,E1 1431.374,E2 1431.374} C_VEL
LIN {X 0,Y 10.957,Z 795.875,A -85,B 0,C 180,E1 1377.146,E2 1377.146} C_VEL
LIN {X 0,Y 11.138,Z 796.189,A -85,B 0,C 180,E1 1349.999,E2 1349.999} C_VEL
LIN {X 0,Y 20.688,Z 794.409,A -85,B 0,C 180,E1 1274.854,E2 1274.854} C_VEL
LIN {X 0,Y 41.009,Z 790.615,A -85,B 0,C 180,E1 1258.387,E2 1258.387} C_VEL
LIN {X 0,Y 61.427,Z 785.12,A -85,B 0,C 180,E1 1253.161,E2 1253.161} C_VEL
LIN {X 0,Y 65.554,Z 783.757,A -85,B 0,C 180,E1 1252.476,E2 1252.476} C_VEL
LIN {X 0,Y 54.43,Z 786.622,A -85,B 0,C 180,E1 1249.434,E2 1249.434} C_VEL
LIN {X 0,Y 45.975,Z 788.577,A -85,B 0,C 180,E1 1247.472,E2 1247.472} C_VEL
LIN {X 0,Y 29.71,Z 791.568,A -85,B 0,C 180,E1 1246.261,E2 1246.261} C_VEL
LIN {X 0,Y 18.429,Z 792.943,A -85,B 0,C 180,E1 1242.637,E2 1242.637} C_VEL
LIN {X 0,Y 14.841,Z 793.195,A -85,B 0,C 180,E1 1238.285,E2 1238.285} C_VEL
LIN {X 0,Y 7.637,Z 793.517,A -85,B 0,C 180,E1 1129.115,E2 1129.115} C_VEL
LIN {X 0,Y 25.449,Z 792.378,A -85,B 0,C 180,E1 1090.836,E2 1090.836} C_VEL
LIN {X 0,Y 25.834,Z 792.351,A -85,B 0,C 180,E1 1090.381,E2 1090.381} C_VEL
LIN {X 0,Y 5.219,Z 794.622,A -85,B 0,C 180,E1 1063.293,E2 1063.293} C_VEL
LIN {X 0,Y 2.926,Z 794.942,A -85,B 0,C 180,E1 989.996,E2 989.996} C_VEL
LIN {X 0,Y 20.232,Z 793.147,A -85,B 0,C 180,E1 891.468,E2 891.468} C_VEL
LIN {X 0,Y 26.162,Z 792.265,A -85,B 0,C 180,E1 889.529,E2 889.529} C_VEL
LIN {X 0,Y 14.841,Z 793.195,A -85,B 0,C 180,E1 878.285,E2 878.285} C_VEL
LIN {X 0,Y 13.153,Z 795.191,A -85,B 0,C 180,E1 874.913,E2 874.913} C_VEL
LIN {X 0,Y 13.153,Z 875,A -85,B 0,C 180,E1 874.913,E2 874.913} C_VEL
LIN {X 0,Y 13.153,Z 875,A -85,B 0,C 180,E1 874.913,E2 874.913}

QRS_NEXT_CUT()

QRS_NEXT()
QRS_HOME()

END
